// TIA Portal V18 export
DATA_BLOCK "!!instanceOf-00_Push-Button_Input$$"   // DB35, F_DB
// stored: InstanceOfName 00_Push-Button_Input, InstanceOfType FB
"00_Push-Button_Input"
   // VAR_INPUT
   //    Bypass_ET200 : Bool;
   //    IN_1 : Bool;
   //    IN_2 : Bool;
   //    IN_3 : Bool;
   //    IN_4 : Bool;
   //    ON_Tristate : Bool;
   //    NormOpenDiag : Bool;
   //    ON_Lamp : Bool;
   //    RESET : Bool;
   //    REAC_DELAY { ExternalWritable := 'False'} : Time;
   //    BLINK_CYCLE_TIME : Time;
   //    ON_TIME : Time;
   // END_VAR
   // VAR_OUTPUT
   //    OUT_1 : Bool;
   //    OUT_2 : Bool;
   //    OUT_3 : Bool;
   //    OUT_4 : Bool;
   //    Diag_1 : Bool;
   //    Diag_2 : Bool;
   //    Diag_3 : Bool;
   //    Diag_4 : Bool;
   //    Lamp_1 : Bool;
   //    Lamp_2 : Bool;
   //    Lamp_3 : Bool;
   //    Lamp_4 : Bool;
   // END_VAR
   // VAR
   //    TON_1 { ExternalWritable := 'False'} : TON;
   //    TON_2 { ExternalWritable := 'False'} : TON;
   //    TON_3 { ExternalWritable := 'False'} : TON;
   //    TON_4 { ExternalWritable := 'False'} : TON;
   //    TOF_Lamp1 : TOF;
   //    TOF_Lamp2 : TOF;
   //    TOF_Lamp3 : TOF;
   //    TOF_Lamp4 : TOF;
   //    PRESSED_1 : Bool;
   //    PRESSED_2 : Bool;
   //    PRESSED_3 : Bool;
   //    PRESSED_4 : Bool;
   //    s_IN_1_P : Bool;
   //    s_IN_2_P : Bool;
   //    s_IN_3_P : Bool;
   //    s_IN_4_P : Bool;
   //    s_IN_1_N : Bool;
   //    s_IN_2_N : Bool;
   //    s_IN_3_N : Bool;
   //    s_IN_4_N : Bool;
   //    DUTY_CYCLE : Time;
   // END_VAR
BEGIN
END_DATA_BLOCK
